PROGRAM OPCUA_Controller
VAR
END_VAR

END_PROGRAM

(* stored: Version 1.1.0.1, ProductVersion 3.1.4022.18
   POU OPCUA_Controller: Id {f5b49519-bcb1-42c8-b86d-25a996ac6a0b}, SpecialFunc None *)
